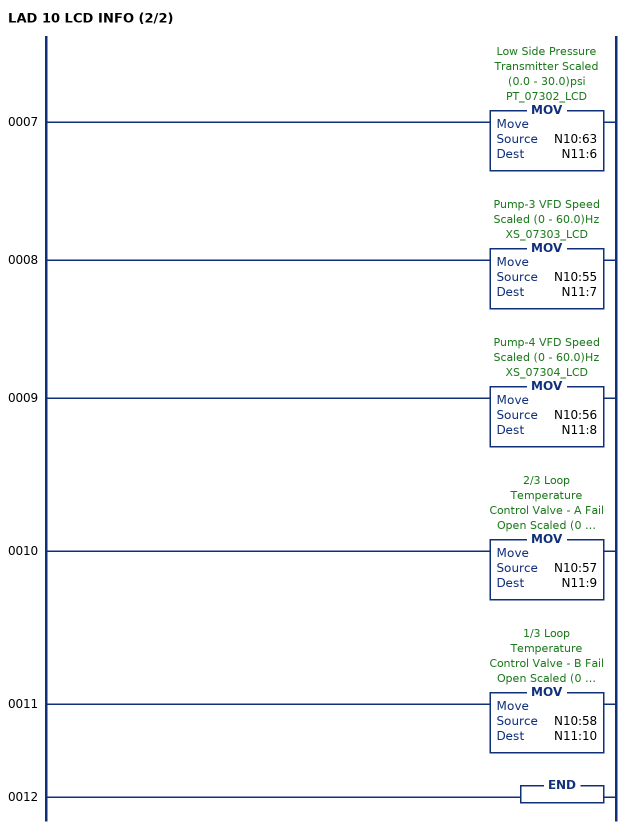
% Rung: 7 %
SOR MOV N10:63 N11:6 EOR
%   N10:63  PT_07302  "Low Side Pressure Transmitter Scaled (0.0 - 30.0)psi" %
%   N11:6  PT_07302_LCD  "Low Side Pressure Transmitter Scaled (0.0 - 30.0)psi" %
% Rung: 8 %
SOR MOV N10:55 N11:7 EOR
%   N10:55  XS_07303  "Pump-3 VFD Speed Scaled (0 - 60.0)Hz" %
%   N11:7  XS_07303_LCD  "Pump-3 VFD Speed Scaled (0 - 60.0)Hz" %
% Rung: 9 %
SOR MOV N10:56 N11:8 EOR
%   N10:56  XS_07304  "Pump-4 VFD Speed Scaled (0 - 60.0)Hz" %
%   N11:8  XS_07304_LCD  "Pump-4 VFD Speed Scaled (0 - 60.0)Hz" %
% Rung: 10 %
SOR MOV N10:57 N11:9 EOR
%   N10:57  TCV_07301A  "2/3 Loop Temperature Control Valve - A Fail Open Scaled (0 - 100.0)%" %
%   N11:9  TCV_07301A_LCD  "2/3 Loop Temperature Control Valve - A Fail Open Scaled (0 - 100.0)%" %
% Rung: 11 %
SOR MOV N10:58 N11:10 EOR
%   N10:58  TCV_07301B  "1/3 Loop Temperature Control Valve - B Fail Open Scaled (0 - 100.0)%" %
%   N11:10  TCV_07301B_LCD  "1/3 Loop Temperature Control Valve - B Fail Open Scaled (0 - 100.0)%" %
% Rung: 12 %
SOR END EOR

OTHER DOCUMENTED ADDRESSES
  B3:0/3  CALCULATE_TEMP_SP
  B3:0/7  TEMP_PID_CLOSE_OK  "TEMPERATURE PID ALLOWED TO CLOSE IN AUTO"
  B3:0/10  HUMID_MAN_OVERRIDE  "Humidifier PID MAN Mode OVERRIDE (1=MAN MODE OVERRIDE, 0=Normal AUTO/MAN Operation)"
  B3:0/11  AIR_FLOW_PID_MANUAL  "Air Flow PID Manual Mode (1 = MAN, 0 = AUTO)"
  B3:0/12  AF_PID_HOLD_OVERRIDE
  B3:1/3  COOL_COIL_PID_MANUAL  "Cooling Coil PID Manual Mode (1=MAN, 0=AUTO)"
  B3:1/5  FLOW_PID_MAN
  B3:1/9  PID_HOLD_OVERRIDE
  B3:1/10  PID_OFF_OVERRIDE
  B3:1/13  COOLING_PID_BIAS_EN  "Cooling Coil PID Setpoint BIAS Enabled"
  B3:3/1  NCW_PUMP_LD_LG  "1=NCW Pump 5 LEAD, NCW Pump 6 LAG 0=NCW Pump 6 LEAD, NCW Pump 5 LAG"
  B3:3/5  ENTHALPY_SR
  B3:3/13  LAD_11_ENABLE
  B3:3/14  LAD_12_ENABLE
  DFILE:0  "OUTPUT"
  DFILE:1  "INPUT"
  DFILE:2  "STATUS"
  DFILE:3  "BINARY"
  DFILE:4  "TIMER"
  DFILE:5  "COUNTER"
  DFILE:6  "CONTROL"
  DFILE:7  "INTEGER"
  DFILE:8  "FLOAT"
  DFILE:9  "PID"
  DFILE:10  "DATA"
  DFILE:11  "LCD DATA"
  DFILE:12  "TT - DATA Temperature Values"
  DFILE:13  "ENT - DATA Entahalpy constants"
  DFILE:14  "AVG TIMERS"
  DFILE:15  "AVG DATA"
  DFILE:16  "AVG FLOAT"
  F8:0  AIR_TEMP_DEC
  F8:1  RETURN_AIR_DEC
  F8:3  ENT_CAL_VAR_1
  F8:4  ENT_CAL_CONST_1
  F8:5  ENT_CALC_VAR_2
  F8:6  ENT_CALC_CONST_2
  F8:7  ENT_CAL_VAR_3
  F8:8  ENT_CAL_CONST_3
  F8:9  ENT_CAL_CONST_4
  F8:10  ENT_CAL_CONST_5
  F8:11  ENTHALPY
  F8:19  RETURN_AIR_ENT
  F8:20  RETURN_VARIABLE
  F8:21  OUTSIDE_AIR_ENT
  F16:1  AVG_DATA_SUM_CH_1
  F16:2  AVG_DATA_SUM_CH_2
  F16:3  AVG_DATA_SUM_CH_3
  F16:4  AVG_DATA_SUM_CH_4
  F16:5  AVG_DATA_SUM_CH_5
  F16:6  AVG_DATA_SUM_CH_6
  F16:7  AVG_DATA_SUM_CH_7
  F16:8  AVG_DATA_SUM_CH_8
  F16:9  AVG_DATA_SUM_CH_9
  F16:10  AVG_DATA_SUM_CH_10
  F16:11  AVG_DATA_SUM_CH_11
  F16:12  AVG_DATA_SUM_CH_12
  F16:13  AVG_DATA_SUM_CH_13
  F16:14  AVG_DATA_SUM_CH_14
  F16:15  AVG_DATA_SUM_CH_15
  F16:16  AVG_DATA_SUM_CH_16
  F16:17  AVG_DATA_SUM_CH_17
  F16:18  AVG_DATA_SUM_CH_18
  F16:19  AVG_DATA_SUM_CH_19
  I:1.1  FT_08367_RAW
  I:3.0  DM_16801_INRAW
  I:3.1  DM_16805A_INRAW
  I:3.2  TT_16351
  I:3.3  MT_16351
  I:4.2  TT_16353
  I:4.3  MT_16353
  I:5.0  TT_16354
  I:5.1  MT_16354
  I:5.2  TT_16355
  I:5.3  MT_16355
  I:6.0  TT_16356
  I:6.1  MT_16356
  I:6.2  TT_16357
  I:6.3  MT_16357
  I:7.0  TT_16358
  I:7.1  MT_16358
  I:7.2  TT_16327B
  I:7.3  "Spare"
  JSR  
  N10:0  SUPPLY_TEMP_DELTA_SP  "T-3 - T1 Delta Setpoint (deg F/10) xxx.x deg F (Tertiary Supply T - Secondary Supply T)"
  N10:1  TEMP_SP_HOLDER  "Tertiary Loop Supply Temperature Setpoint Temporary Holder"
  N10:5  TT2_TT1_CLOSE_SP  "When TT-2 minus TT-1 is less than this Setpoint (14.0 degF) then TCV will be allowed to close"
  N10:6  TT2_MINUS_TT1  "TT2 - TT1 SEC. CHWR minus SEC. CHWS"
  N10:9  COOL_PID_SP_TEMP  "Temporary Setpoint Holder"
  N10:15  TCV_16826  "Chilled Water Control Valve Scaled 0-100%"
  N10:16  TT_16801_PV  "Outside Air Temperature Scaled for PID"
  N10:19  FT_08367
  N10:25  XS_0916X_1_S  "Cooling Tower Fan Speed Scaled 0-60.0 Hz"
  N10:26  TT_16805_PV  "Return Air Temperature Scaled for PID"
  N10:30  TT_09175_S_LIMITS  "Nitride Cooling Water Supply Temperature Highest with Limits"
  N10:31  TT_09175_S_LO_LIMIT
  N10:33  XS_0916X_1_LO_SPEED
  N10:34  XS_0916X_1_HI_SPEED
  N10:36  TT_16817A_PV
  N10:37  TT_16817B_PV
  N10:42  TT_16817A
  N10:43  TT_16817B
  N10:46  TT_16825_PV
  N10:65  TT_3_PID  "T-3 (TT08367C) Tertiary CHW Supply Temperature Scaled for PID"
  N10:70  DM_16801_IN
  N10:71  DM_16805A_IN
  N10:76  TT_16826_PV
  N10:86  DM_16801_IN_PV
  N10:87  DM_16805A_IN_PV
  N10:96  TT_16845_PV
  N10:97  TCV_16826_CV
  N10:98  COOLING_COIL_PID_SP
  N10:99  COOLING_PID_SP_ENTER
  N10:123  COOLING_PID_WW_P  "Cooling PID WW Proportional Parameter"
  N10:124  COOLING_PID_WW_I  "Cooling PID WW Integral Parameter"
  N10:125  COOLING_PID_WW_D  "Cooling PID WW Derivative Parameter"
  N10:173  COOLING_PID_WW_TMP_P  "Cooling PID Temporary Proportional Parameter"
  N10:174  COOLING_PID_WW_TMP_I  "Cooling PID Temporary Integral Parameter"
  N10:175  COOLING_PID_WW_TMP_D  "Cooling PID Temporary Derivative Parameter"
  N10:199  REHEAT8_PID_WW_TMP_D
  N11:11  TCV_16833_LCD
  N11:12  TCV_16834_LCD
  N11:13  TCV_16837_LCD
  N11:14  TCV_16838_LCD
  N11:48  LCD_PROTECT_1  "Data Protection Words 0-15"
  N11:49  LCD_PROTECT_2  "Data Protection Words 16-31"
  N11:50  LCD_PROTECT_3  "Data Protection Words 32-47"
  N15:0  AVG_DATA_POINT_IN
  N15:1  AVG_AVG_VALUE_OUT
  N15:2  AVG_INDEX
  N15:201  AVG_RAWDATA_CH_1
  N15:202  AVG_RAWDATA_CH_2
  N15:203  AVG_RAWDATA_CH_3
  N15:204  AVG_RAWDATA_CH_4
  N15:205  AVG_RAWDATA_CH_5
  N15:206  AVG_RAWDATA_CH_6
  N15:207  AVG_RAWDATA_CH_7
  N15:208  AVG_RAWDATA_CH_8
  N15:209  AVG_RAWDATA_CH_9
  N15:210  AVG_RAWDATA_CH_10
  N15:211  AVG_RAWDATA_CH_11
  N15:212  AVG_RAWDATA_CH_12
  N15:213  AVG_RAWDATA_CH_13
  N15:214  AVG_RAWDATA_CH_14
  N15:215  AVG_RAWDATA_CH_15
  N15:216  AVG_RAWDATA_CH_16
  N15:217  AVG_RAWDATA_CH_17
  N15:218  AVG_RAWDATA_CH_18
  N15:219  AVG_RAWDATA_CH_19
  N15:221  AVG_OFFSET_1
  N15:222  AVG_OFFSET_2
  N15:223  AVG_OFFSET_3
  N15:224  AVG_OFFSET_4
  N15:225  AVG_OFFSET_5
  N15:226  AVG_OFFSET_6
  N15:227  AVG_OFFSET_7
  N15:228  AVG_OFFSET_8
  N15:229  AVG_OFFSET_9
  N15:230  AVG_OFFSET_10
  N15:231  AVG_INDEX_RAW_INPUT
  O:4.0  TCV_16826_RAW
  O:4.1  DM_16801_RAW
  O:4.2  DM_16805A_RAW
  O:5.0  TCV_16336
  O:5.1  TCV_16337
  O:6.0  TCV_16338
  O:6.1  XS_EF2_SPEED
  PD9:0  RHC_1_PID
  PD9:3  RHC_4_PID
  PD9:4  RHC_7_PID
  PD9:5  RHC_8_PID
  PD9:9  COOLING_COIL_PID
  PD9:10  HUMIDIFIER_PID
  PD9:11  FLOW_PID
  PFILE:3  "Temperature scaling for enthalpy calc"
  PFILE:4  "Analog Scaling and A larms"
  PFILE:5  "AHU Fan and Damper L ogic"
  PFILE:6  "Tertiary Loop CHWP-2 Control"
  PFILE:7  "Tertiary Loop Pressu re Differential Cont rol"
  PFILE:8  "Reheat Coils Logic"
  PFILE:11  "VFD Flow Control"
  T4:4  ENTHALPY_TIMER  "Enthalpy Timer"
  T4:4/DN  "Humidifier Alarm Timer DN"
  T4:5  RLF_FAN_RUN_FB  "Relief Fan Running Feedback Timer"
  T4:6  PID_OFF_OVERRIDE_TMR
  T4:7  "Fan Running Delay Timer ON"
  T4:8  "Fan Running Delay Timer Off"
  T14:1  AVG_SAMPLE_TMR_CH_1
  T14:2  AVG_SAMPLE_TMR_CH_2
  T14:3  AVG_SAMPLE_TMR_CH_3
  T14:4  AVG_SAMPLE_TMR_CH_4
  T14:5  AVG_SAMPLE_TMR_CH_5
  T14:6  AVG_SAMPLE_TMR_CH_6
  T14:7  AVG_SAMPLE_TMR_CH_7
  T14:8  AVG_SAMPLE_TMR_CH_8
  T14:9  AVG_SAMPLE_TMR_CH_9
  T14:10  AVG_SAMPLE_TMR_CH_10
  T14:11  AVG_SAMPLE_TMR_CH_11
  T14:12  AVG_SAMPLE_TMR_CH_12
  T14:13  AVG_SAMPLE_TMR_CH_13
  T14:14  AVG_SAMPLE_TMR_CH_14
  T14:15  AVG_SAMPLE_TMR_CH_15
  T14:16  AVG_SAMPLE_TMR_CH_16
  T14:17  AVG_SAMPLE_TMR_CH_17
  T14:18  AVG_SAMPLE_TMR_CH_18
  T14:19  AVG_SAMPLE_TMR_CH_19
  U:3  "Enthalpy Sub-Routine"

DATA TABLE (non-zero values as saved)
DATA B3
% B3:0 % 0X0188 0XA026 0X0067 0X7FC3 0X0000 0X0002 0X0000 0X0000 0X0000 0X0000
DATA T4
% .PRE .ACC %
% T4:0 % 30 0
% T4:1 % 3600 2899
% T4:2 % 3600 2808
% T4:3 % 10 0
% T4:4 % 600 313
% T4:5 % 10 0
% T4:6 % 90 0
% T4:7 % 1 0
% T4:8 % 2 2
% T4:40 % 12 0
% T4:42 % 2 0
% T4:43 % 20 0
% T4:44 % 1 0
% T4:45 % 2 2
% T4:46 % 3 3
% T4:50 % 12 0
% T4:52 % 2 0
% T4:53 % 20 0
% T4:54 % 1 1
% T4:55 % 2 0
% T4:56 % 3 0
DATA C5
% .PRE .ACC %
% C5:0 % 32000 5858
% C5:1 % 32000 2640
DATA F8
% F8:0 % 71.8
DATA N10
% N10:0 % 10 762 2739 8061 100 140 -13 11734 0 650
% N10:10 % 0 0 0 0 0 343 9481 2684 1800 0
% N10:20 % 100 0 0 0 0 150 7963 0 700 0
% N10:30 % 870 870 323 200 600 0 7234 0 700 0
% N10:40 % 1791 0 868 868 0 0 7201 4408 700 0
% N10:50 % 1306 0 0 0 0 295 295 329 0 0
% N10:60 % 0 0 606 151 54 12647 0 0 0 0
% N10:70 % 669 0 0 0 0 0 6727 8528 700 0
% N10:80 % 0 0 0 0 0 0 6567 8634 700 0
% N10:90 % 5 22 10 3 11 0 6630 5617 550 700
% N10:100 % 5 22 10 3 11 0 0 0 0 0
% N10:120 % 0 0 0 5 15 0 3 11 0 3
% N10:130 % 11 0 3 11 0 3 11 0 0 0
% N10:140 % 0 0 0 0 3 11 0 3 11 0
% N10:170 % 0 0 0 5 15 0 3 11 0 3
% N10:180 % 11 0 3 11 0 3 11 0 0 0
% N10:190 % 0 0 0 0 3 11 0 3 11 0
DATA N11
% N11:0 % 100 0 323 1791 1306 606 151 295 295 329
% N11:10 % 0 0 0 41 54 0 0 0 0 0
DATA N12
% N12:0 % -50 50 150 250 350 450 550 650 750 850
% N12:10 % 950 1050 1150 1250 1350 1450 1550 1650 1750 0
